PROGRAM PRG_Test
VAR
END_VAR


	TcUnit.RUN_IN_SEQUENCE ();

END_PROGRAM

(* stored: Version 1.1.0.1
   POU PRG_Test: Id {f3067e18-a8df-4ccb-9920-df5f52e60274}, SpecialFunc None *)
